(* IEC 61131-3 sources: windowtracking/src/lib/Events, 3 files *)

(* ---- EventStatus.st ---- *)
NAMESPACE Simatic.Ax.WindowTracking.Events

    TYPE
        EventStatus : (Undefined, Finished, Error, NullReference) := Undefined;
    END_TYPE

END_NAMESPACE

(* ---- VirtualTrigger.st ---- *)
USING Simatic.Ax.WindowTracking.VirtualTrigger;
NAMESPACE Simatic.Ax.WindowTracking.Events
    CLASS VirtualTrigger IMPLEMENTS IVirtualTrigger

        VAR PUBLIC
            Position : DINT;
            Id : UINT;
            EventHandler : ITriggerEvent;
        END_VAR

        VAR PROTECTED
            _isActiavted : BOOL;
        END_VAR

        METHOD PUBLIC ActivateEvent : EventStatus
            VAR_INPUT
                tw : ITransportWindow;
            END_VAR
            IF EventHandler <> NULL THEN
                ActivateEvent := EventHandler.Action(te := THIS, tw := tw);
                RETURN;
            ELSE
                ActivateEvent := Eventstatus#NullReference;
            END_IF;

        END_METHOD

        METHOD PUBLIC IsActivated
            ;
        END_METHOD

        METHOD PUBLIC GetID : UINT
            GetID := Id;
        END_METHOD

        METHOD PUBLIC GetPosition : DINT
            GetPosition := Position;
        END_METHOD

        METHOD PUBLIC IsEnabled : BOOL
            IsEnabled := TRUE;
        END_METHOD

    END_CLASS
END_NAMESPACE

(* ---- VirtualTriggerList.st ---- *)
NAMESPACE Simatic.Ax.WindowTracking.VirtualTrigger
    CLASS TriggerPoints
        VAR PUBLIC

        END_VAR
        VAR PROTECTED
            _triggerPointList : ARRAY[UINT#0..BUF_SIZE - UINT#1] OF IVirtualTrigger;
            _count : UINT;
        END_VAR

        VAR CONSTANT
            BUF_SIZE : UINT := UINT#100;
        END_VAR

        METHOD PUBLIC Add : BOOL
            VAR_INPUT
                tp : IVirtualTrigger;
            END_VAR
            IF (_count < BUF_SIZE) THEN
                _triggerPointList[_count] := tp;
                _count := _count + UINT#1;
            ELSE
                Add := FALSE;
            END_IF;
        END_METHOD

        METHOD PUBLIC Count : UINT
            Count := _count;
        END_METHOD

        METHOD PUBLIC GetTriggerPoint : IVirtualTrigger
            VAR_INPUT
                Id : UINT;
            END_VAR
            VAR_TEMP
                i : UINT;
            END_VAR
            FOR i := UINT#0 TO THIS.Count() - UINT#1 DO
                IF (_triggerPointList[i].GetId() = Id) THEN
                    GetTriggerPoint := _triggerPointList[i];
                    RETURN;
                END_IF;
            END_FOR;
            GetTriggerPoint := NULL;
        END_METHOD
    END_CLASS

END_NAMESPACE
